# EPICS autosave request: support/sscan/2-6-4/sscanApp/Db/scan_settings.req
# FILE... scan_settings.req
# USAGE.. scan.db fields autosave'd.
$(P)$(S).AAWAIT
$(P)$(S).FLNK
$(P)$(S).NPTS
$(P)$(S).ACQT
$(P)$(S).ACQM
$(P)$(S).PASM
$(P)$(S).BSPV
$(P)$(S).BSCD
$(P)$(S).BSWAIT
$(P)$(S).ASPV
$(P)$(S).ASCD
$(P)$(S).ASWAIT
$(P)$(S).T1PV
$(P)$(S).T1CD
$(P)$(S).T2PV
$(P)$(S).T2CD
$(P)$(S).T3PV
$(P)$(S).T3CD
$(P)$(S).T4PV
$(P)$(S).T4CD
$(P)$(S).P1PV
$(P)$(S).R1PV
$(P)$(S).P1SM
$(P)$(S).P1SP
$(P)$(S).P1EP
$(P)$(S).P1AR
$(P)$(S).P2PV
$(P)$(S).R2PV
$(P)$(S).P2SM
$(P)$(S).P2SP
$(P)$(S).P2EP
$(P)$(S).P2AR
$(P)$(S).P3PV
$(P)$(S).R3PV
$(P)$(S).P3SM
$(P)$(S).P3SP
$(P)$(S).P3EP
$(P)$(S).P3AR
$(P)$(S).P4PV
$(P)$(S).R4PV
$(P)$(S).P4SM
$(P)$(S).P4SP
$(P)$(S).P4EP
$(P)$(S).P4AR
$(P)$(S).PDLY
$(P)$(S).DDLY
$(P)$(S).REFD
$(P)$(S).AWCT
$(P)$(S).A1PV
$(P)$(S).A1CD
$(P)$(S).D01PV
$(P)$(S).D02PV
$(P)$(S).D03PV
$(P)$(S).D04PV
$(P)$(S).D05PV
$(P)$(S).D06PV
$(P)$(S).D07PV
$(P)$(S).D08PV
$(P)$(S).D09PV
$(P)$(S).D10PV
$(P)$(S).D11PV
$(P)$(S).D12PV
$(P)$(S).D13PV
$(P)$(S).D14PV
$(P)$(S).D15PV
$(P)$(S).D16PV
$(P)$(S).D17PV
$(P)$(S).D18PV
$(P)$(S).D19PV
$(P)$(S).D20PV
$(P)$(S).D21PV
$(P)$(S).D22PV
$(P)$(S).D23PV
$(P)$(S).D24PV
$(P)$(S).D25PV
$(P)$(S).D26PV
$(P)$(S).D27PV
$(P)$(S).D28PV
$(P)$(S).D29PV
$(P)$(S).D30PV
$(P)$(S).D31PV
$(P)$(S).D32PV
$(P)$(S).D33PV
$(P)$(S).D34PV
$(P)$(S).D35PV
$(P)$(S).D36PV
$(P)$(S).D37PV
$(P)$(S).D38PV
$(P)$(S).D39PV
$(P)$(S).D40PV
$(P)$(S).D41PV
$(P)$(S).D42PV
$(P)$(S).D43PV
$(P)$(S).D44PV
$(P)$(S).D45PV
$(P)$(S).D46PV
$(P)$(S).D47PV
$(P)$(S).D48PV
$(P)$(S).D49PV
$(P)$(S).D50PV
$(P)$(S).D51PV
$(P)$(S).D52PV
$(P)$(S).D53PV
$(P)$(S).D54PV
$(P)$(S).D55PV
$(P)$(S).D56PV
$(P)$(S).D57PV
$(P)$(S).D58PV
$(P)$(S).D59PV
$(P)$(S).D60PV
$(P)$(S).D61PV
$(P)$(S).D62PV
$(P)$(S).D63PV
$(P)$(S).D64PV
$(P)$(S).D65PV
$(P)$(S).D66PV
$(P)$(S).D67PV
$(P)$(S).D68PV
$(P)$(S).D69PV
$(P)$(S).D70PV
